
FUNCTION CB_sel_dword : DINT


TITLE = ' Binary selection on 2 variables '
VERSION : '1.0'
AUTHOR  : CB
NAME    : selDword
FAMILY  : TNI

VAR_INPUT
    G : BOOL;
    IN0 : DINT ;
    IN1 : DINT ;

END_VAR

BEGIN

CB_sel_dword := SEL(G:= G, IN0 := IN0, IN1 := IN1);

END_FUNCTION
